FUNCTION_BLOCK FB_SafetySignalsSZPCo
VAR_INPUT
	ErrorAck		: BOOL; //Summarized from all reset safety buttons located within safety zone
END_VAR
VAR_OUTPUT
	TwinSafeError	: BOOL; //Error in FB or Com in TwinSafe
	TwinSafeOK		: BOOL; //Summary of Safety zone inputs
END_VAR
VAR_IN_OUT
	SZPCoSignals	:	ST_ProBoxSafetySZPCo;
END_VAR
VAR	
	i			: INT;
END_VAR

//Indicate that an error exit with blinking blue lamp on cabinet. 
IF (SZPCoSignals.Inputs.ComErr OR SZPCoSignals.Inputs.FBErr) THEN
	TwinSafeError := TRUE;
ELSE 
	TwinSafeError := FALSE;
END_IF

TwinSafeOK := SZPCoSignals.Inputs.SafetyZoneOk AND NOT TwinSafeError;

//Pass on pushbutton and pass on to Safety
SZPCoSignals.Outputs.ErrorAck := ErrorAck;

END_FUNCTION_BLOCK

(* stored: Version 1.1.0.1, ProductVersion 3.1.4024.9
   POU FB_SafetySignalsSZPCo: Id {eb0a1f19-0a53-4993-afa6-e4e35ef074e5}, SpecialFunc None *)
